Universal Robots PolyScope program: 34-trigger_reduced_mode_feature.urp

ProgramRoot directory=/programs/usbdisk; kinematics=(a=[0.00023, -0.38811, -0.39243, -0.00016, 0.00019, 0], d=[0.08925, 195.22769, -194.66383, -0.45311, 0.09509, 0.08264], alpha=[1.57049, -0.00089, 0.00686, 1.56999, -1.56996, 0], deltaTheta=[-0.00001, -0.41907, 0.4289, -6.29306, -0.00007, 0], status=notLinearised); lastSavedInVersion=(project__name=Polyscope, major__version=3, minor__version=1, svn__revision=17141, build__date=Mar 06 2015, 07:52:30); name=34-trigger_reduced_mode_feature; programVersion=(project__name=Polyscope, major__version=3, minor__version=1, svn__revision=17141, build__date=Mar 06 2015, 07:52:30); robotEnvironmentFileName=feature; serialNumberRobot=2014350456
  MainProgram cartesianAcceleration=1.2; cartesianSpeed=0.25; jointAcceleration=1.3962634015954636; jointSpeed=1.0471975511965976; sharedProcessMoveBlendRadius=0.025; motionType=JOINT_SPACE
    Move cartesianAcceleration=1.2; cartesianSpeed=0.25; jointAcceleration=1.3962634015954636; jointSpeed=1.0471975511965976; sharedProcessMoveBlendRadius=0.025; motionType=CARTESIAN_SPACE
      Waypoint blendRadius=0.05; cartesianAcceleration=1.2; cartesianSpeed=0.25; jointAcceleration=1.3962634015954636; jointSpeed=1.0471975511965976; nextMotionTime=2.0; stoppoint=true; useSharedBlendParameter=true; useSharedParameters=true; outputFlangePose=(pos=(x=-0.07536091946476275, y=0.20456325259765754, z=0.3713647811153902), rot=(x=2.2860240074678044, y=-2.075320194966536, z=0.07862301514892728)); position=TCP in base x=-75.349 y=204.562 z=371.352 mm, rx=2.286 ry=-2.0754 rz=0.0787 rad; joints [-220.62, -47.144, -124.472, -101.266, 93.545, 133.688] deg; positionType=FIXED_POSITION; waypointPoseInFeatureCoordinates=(pos=(x=-0.0753493159766643, y=0.2045618775146442, z=0.3713522738010673), rot=(x=2.2859912252735977, y=-2.075391354330745, z=0.0786962723113226)); name=路点_1
      Waypoint blendRadius=0.05; cartesianAcceleration=1.2; cartesianSpeed=0.25; jointAcceleration=1.3962634015954636; jointSpeed=1.0471975511965976; nextMotionTime=2.0; stoppoint=true; useSharedBlendParameter=true; useSharedParameters=true; outputFlangePose=(pos=(x=-0.3862808410612096, y=0.587543446928109, z=0.4101295038909787), rot=(x=2.152315254142266, y=-2.2128392761425943, z=-0.11027197465442934)); position=TCP in base x=-386.294 y=587.551 z=410.101 mm, rx=2.1524 ry=-2.2128 rz=-0.1102 rad; joints [-227.992, -118.456, -58.239, -89.375, 93.545, 133.687] deg; positionType=FIXED_POSITION; waypointPoseInFeatureCoordinates=(pos=(x=-0.3862936358287604, y=0.5875509185211385, z=0.4101006419699886), rot=(x=2.152386688518448, y=-2.2128377831054413, z=-0.11023383767056169)); name=路点_2
